// TIA Portal V15.1 export
// export: Created 2024-05-17T05:38:33.3667572Z, ExportSetting WithDefaults, DisplayName Totally Integrated Automation Portal, DisplayVersion V15.1 Update 5, DisplayName TIA Portal Openness, DisplayVersion V15.1 Update 5, DisplayName SINAMICS Startdrive Advanced, DisplayVersion V15.1, DisplayName G130, G150, S120, S150, SINAMICS MV, S210, DisplayVersion V15.1, DisplayName G110M, G120, G120C, G120D, G120P, DisplayVersion V15.1, DisplayName STEP 7 Professional, DisplayVersion V15.1 Update 5, DisplayName STEP 7 Safety, DisplayVersion V15.1, DisplayName WinCC Professional, DisplayVersion V15.1 Update 5, DisplayName SIMATIC Visualization Architect, DisplayVersion V15.1
FUNCTION_BLOCK "LProcDO_NoFbk"   // FB1711, FBD
TITLE = LProcDO_NoFbk
{ S7_Optimized_Access := 'FALSE' }
AUTHOR : VCC
FAMILY : ProcEq
NAME : DONoFbk
VERSION : 0.1
// ================================================================================
// This module converts the signal 0-100% to digital commands Open and Close to 
// steer in position a valve or damper equipped with a motor.
// There is no feedback, the controller is operating with a time.
// Detections Open/Close may be connected to the controller to check the correct 
// opening and closing of the valve or damper.
// ================================================================================
// stored: AutoNumber false, IsIECCheckEnabled false, SetENOAutomatically False, UDAEnableTagReadback false
   VAR_INPUT
      I_CYCLE { ExternalAccessible := 'False'; ExternalVisible := 'False'; ExternalWritable := 'False'} : Time;   // Sample time
      H_PULSE_TM : Time;   // Minimum Pulse Time
      H_BREAK_TM : Time;   // Minimum Break Time
      H_MTR_TM : Time;   // Motor manipulated time value
      I_SP : Real;   // Set-point Input
      H_DEADB_W : Real;   // Slave: Deadband width
      I_COM_RST { ExternalAccessible := 'False'; ExternalVisible := 'False'; ExternalWritable := 'False'} : Bool;   // Initialising reset of controller
   END_VAR
   VAR_OUTPUT
      O_PosFbk { ExternalAccessible := 'False'; ExternalVisible := 'False'; ExternalWritable := 'False'} : Real;   // Output Feedback Position
      O_Set { ExternalAccessible := 'False'; ExternalVisible := 'False'; ExternalWritable := 'False'} : Bool;   // DO output Set
      O_Reset { ExternalAccessible := 'False'; ExternalVisible := 'False'; ExternalWritable := 'False'} : Bool;   // DO output Reset
   END_VAR
   VAR
      DO_Controller { ExternalAccessible := 'False'; ExternalVisible := 'False'; ExternalWritable := 'False'; S7_SetPoint := 'True'} : CONT_S;
   END_VAR
BEGIN

REGION Network 1: **** 5.2 - Equations - Flow Equations **** Activate DO controller
   // Activate DO controller
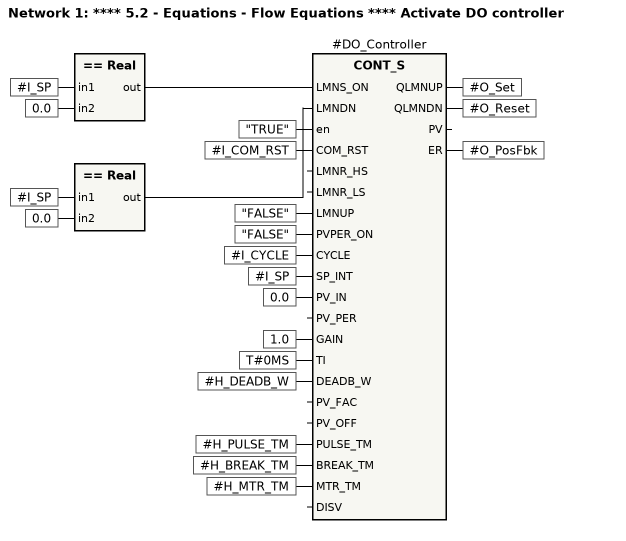
   IF "TRUE" THEN
       #DO_Controller(LMNS_ON := #I_SP = 0.0,   // CONT_S
                      LMNDN := #I_SP = 0.0,
                      COM_RST := #I_COM_RST,
                      LMNUP := "FALSE",
                      PVPER_ON := "FALSE",
                      CYCLE := #I_CYCLE,
                      SP_INT := #I_SP,
                      PV_IN := 0.0,
                      GAIN := 1.0,
                      TI := T#0MS,
                      DEADB_W := #H_DEADB_W,
                      PULSE_TM := #H_PULSE_TM,
                      BREAK_TM := #H_BREAK_TM,
                      MTR_TM := #H_MTR_TM,
                      QLMNUP => #O_Set,
                      QLMNDN => #O_Reset,
                      ER => #O_PosFbk);
   END_IF;
END_REGION
END_FUNCTION_BLOCK
